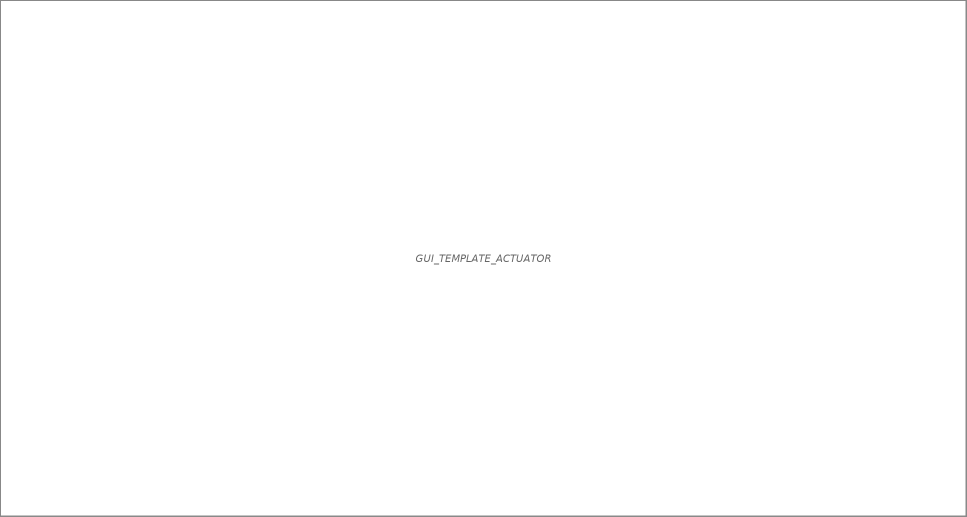
VISUALIZATION GUI_Actuator003  // 967x517
    Frame (0,0 967x517)
        shows GUI_TEMPLATE_ACTUATOR(m_Instance := MAIN.Actuator003)
END_VISUALIZATION

(* stored: Version 1.1.0.1, ProductVersion 3.1.4024.3
   Visu GUI_Actuator003: Id {9d003725-e3dd-4a72-894a-1a5789ec745d} *)
